LIN {X 0,Y 11.902,Z 818.178,A -85,B 0,C 180,E1 -31013.809,E2 -31013.809} C_VEL
LIN {X 0,Y 0.249,Z 818.178,A -85,B 0,C 180,E1 -30870,E2 -30870} C_VEL
LIN {X 0,Y 11.637,Z 818.178,A -85,B 0,C 180,E1 -30727.151,E2 -30727.151} C_VEL
LIN {X 0,Y 17.346,Z 818.178,A -85,B 0,C 180,E1 -30725.832,E2 -30725.832} C_VEL
LIN {X 0,Y 21.805,Z 818.096,A -85,B 0,C 180,E1 -30726.285,E2 -30726.285} C_VEL
LIN {X 0,Y 23.073,Z 821.024,A -85,B 0,C 180,E1 -30726.883,E2 -30726.883} C_VEL
LIN {X 0,Y 26.796,Z 827.658,A -85,B 0,C 180,E1 -30720.613,E2 -30720.613} C_VEL
LIN {X 0,Y 27.089,Z 826.107,A -85,B 0,C 180,E1 -30712.91,E2 -30712.91} C_VEL
LIN {X 0,Y 28.425,Z 821.177,A -85,B 0,C 180,E1 -30698.416,E2 -30698.416} C_VEL
LIN {X 0,Y 31.563,Z 817.637,A -85,B 0,C 180,E1 -30687.882,E2 -30687.882} C_VEL
LIN {X 0,Y 28.79,Z 821.493,A -85,B 0,C 180,E1 -30675.871,E2 -30675.871} C_VEL
LIN {X 0,Y 28.462,Z 822.418,A -85,B 0,C 180,E1 -30673.109,E2 -30673.109} C_VEL
LIN {X 0,Y 27.429,Z 823.083,A -85,B 0,C 180,E1 -30670.442,E2 -30670.442} C_VEL
LIN {X 0,Y 25.047,Z 823.175,A -85,B 0,C 180,E1 -30668.077,E2 -30668.077} C_VEL
LIN {X 0,Y 21.285,Z 822.425,A -85,B 0,C 180,E1 -30666.813,E2 -30666.813} C_VEL
LIN {X 0,Y 16.795,Z 821.066,A -85,B 0,C 180,E1 -30667.552,E2 -30667.552} C_VEL
LIN {X 0,Y 12.429,Z 819.293,A -85,B 0,C 180,E1 -30674.591,E2 -30674.591} C_VEL
LIN {X 0,Y 11.327,Z 818.488,A -85,B 0,C 180,E1 -30683.281,E2 -30683.281} C_VEL
LIN {X 0,Y 11.746,Z 818.178,A -85,B 0,C 180,E1 -30690,E2 -30690} C_VEL
LIN {X 0,Y 22.119,Z 818.086,A -85,B 0,C 180,E1 -30707.533,E2 -30707.533} C_VEL
LIN {X 0,Y 22.768,Z 818.067,A -85,B 0,C 180,E1 -30690,E2 -30690} C_VEL
LIN {X 0,Y 22.014,Z 818.089,A -85,B 0,C 180,E1 -30673.354,E2 -30673.354} C_VEL
LIN {X 0,Y 11.746,Z 818.178,A -85,B 0,C 180,E1 -30690,E2 -30690} C_VEL
LIN {X 0,Y 11.746,Z 818.178,A -85,B 0,C 180,E1 -30690,E2 -30690}

QRS_NEXT_CUT()

QRS_NEXT()
QRS_HOME()

END
